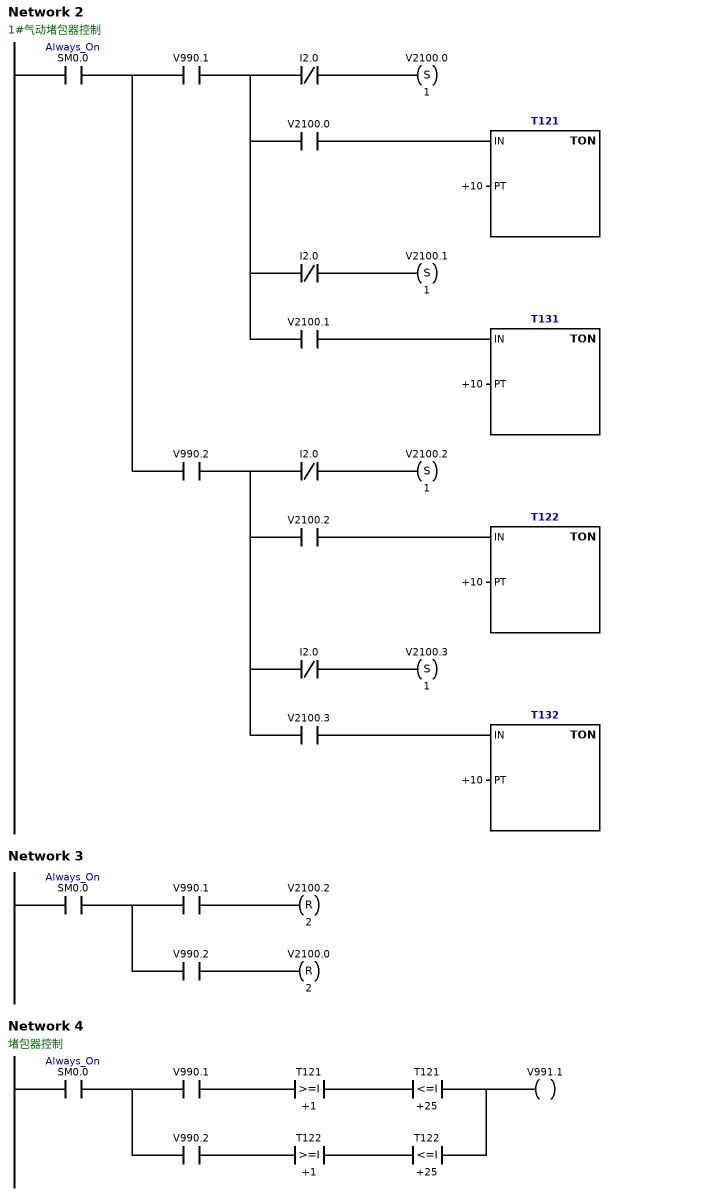
[picture p72: SBR29 networks 2-4]
Network 2
// 1#气动堵包器控制
LD     Always_On:SM0.0
LPS
A      V990.1
LPS
AN     I2.0
S      V2100.0, 1
LRD
A      V2100.0
TON    T121, +10
LRD
AN     I2.0
S      V2100.1, 1
LPP
A      V2100.1
TON    T131, +10
LPP
A      V990.2
LPS
AN     I2.0
S      V2100.2, 1
LRD
A      V2100.2
TON    T122, +10
LRD
AN     I2.0
S      V2100.3, 1
LPP
A      V2100.3
TON    T132, +10
Network 3
LD     Always_On:SM0.0
LPS
A      V990.1
R      V2100.2, 2
LPP
A      V990.2
R      V2100.0, 2
Network 4
// 堵包器控制
LD     Always_On:SM0.0
LD     V990.1
AW>=   T121, +1
AW<=   T121, +25
LD     V990.2
AW>=   T122, +1
AW<=   T122, +25
OLD
ALD
=      V991.1
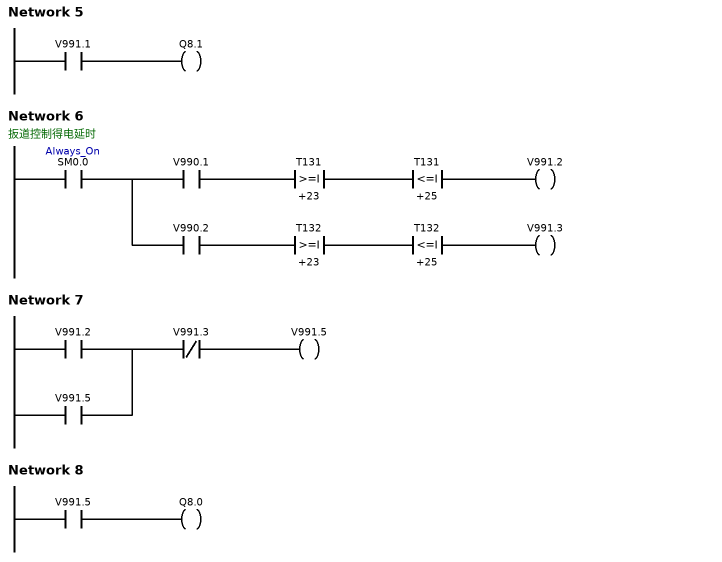
Network 5
LD     V991.1
=      Q8.1
Network 6
// 扳道控制得电延时
LD     Always_On:SM0.0
LPS
A      V990.1
AW>=   T131, +23
AW<=   T131, +25
=      V991.2
LPP
A      V990.2
AW>=   T132, +23
AW<=   T132, +25
=      V991.3
Network 7
LD     V991.2
O      V991.5
AN     V991.3
=      V991.5
Network 8
LD     V991.5
=      Q8.0
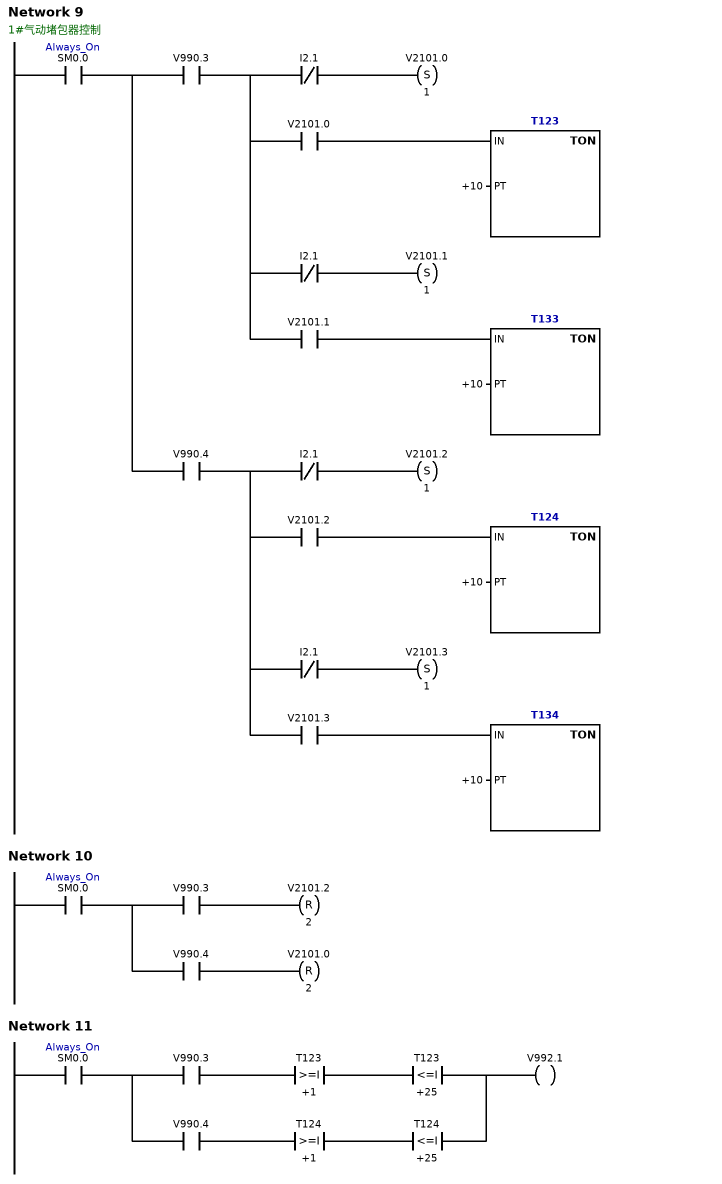
Network 9
// 1#气动堵包器控制
LD     Always_On:SM0.0
LPS
A      V990.3
LPS
AN     I2.1
S      V2101.0, 1
LRD
A      V2101.0
TON    T123, +10
LRD
AN     I2.1
S      V2101.1, 1
LPP
A      V2101.1
TON    T133, +10
LPP
A      V990.4
LPS
AN     I2.1
S      V2101.2, 1
LRD
A      V2101.2
TON    T124, +10
LRD
AN     I2.1
S      V2101.3, 1
LPP
A      V2101.3
TON    T134, +10
Network 10
LD     Always_On:SM0.0
LPS
A      V990.3
R      V2101.2, 2
LPP
A      V990.4
R      V2101.0, 2
Network 11
LD     Always_On:SM0.0
LD     V990.3
AW>=   T123, +1
AW<=   T123, +25
LD     V990.4
AW>=   T124, +1
AW<=   T124, +25
OLD
ALD
=      V992.1
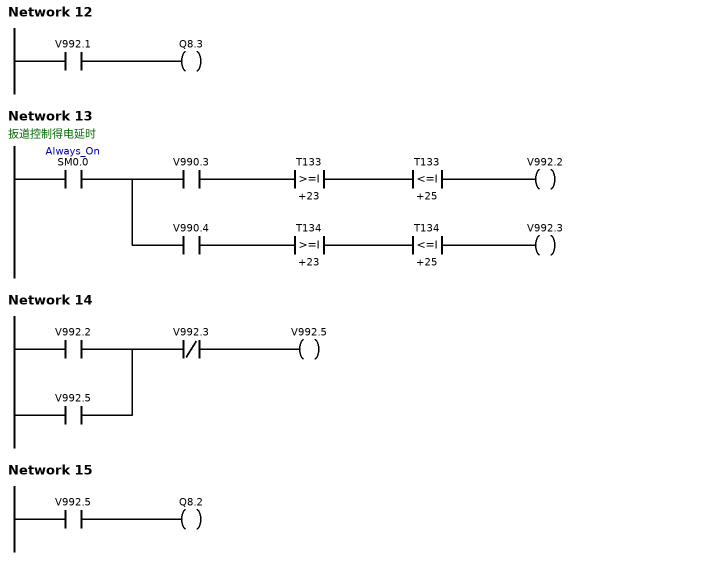
Network 12
LD     V992.1
=      Q8.3
Network 13
// 扳道控制得电延时
LD     Always_On:SM0.0
LPS
A      V990.3
AW>=   T133, +23
AW<=   T133, +25
=      V992.2
LPP
A      V990.4
AW>=   T134, +23
AW<=   T134, +25
=      V992.3
Network 14
LD     V992.2
O      V992.5
AN     V992.3
=      V992.5
Network 15
LD     V992.5
=      Q8.2
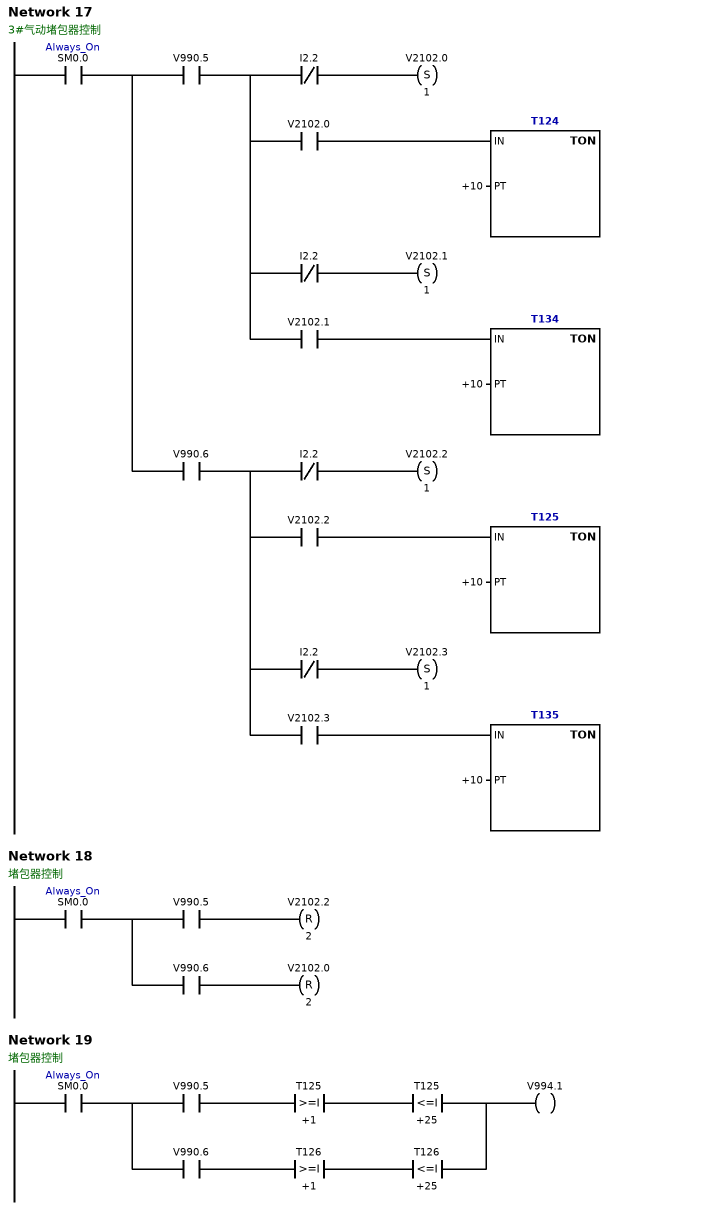
Network 17
// 3#气动堵包器控制
LD     Always_On:SM0.0
LPS
A      V990.5
LPS
AN     I2.2
S      V2102.0, 1
LRD
A      V2102.0
TON    T124, +10
LRD
AN     I2.2
S      V2102.1, 1
LPP
A      V2102.1
TON    T134, +10
LPP
A      V990.6
LPS
AN     I2.2
S      V2102.2, 1
LRD
A      V2102.2
TON    T125, +10
LRD
AN     I2.2
S      V2102.3, 1
LPP
A      V2102.3
TON    T135, +10
Network 18
// 堵包器控制
LD     Always_On:SM0.0
LPS
A      V990.5
R      V2102.2, 2
LPP
A      V990.6
R      V2102.0, 2
Network 19
// 堵包器控制
LD     Always_On:SM0.0
LD     V990.5
AW>=   T125, +1
AW<=   T125, +25
LD     V990.6
AW>=   T126, +1
AW<=   T126, +25
OLD
ALD
=      V994.1
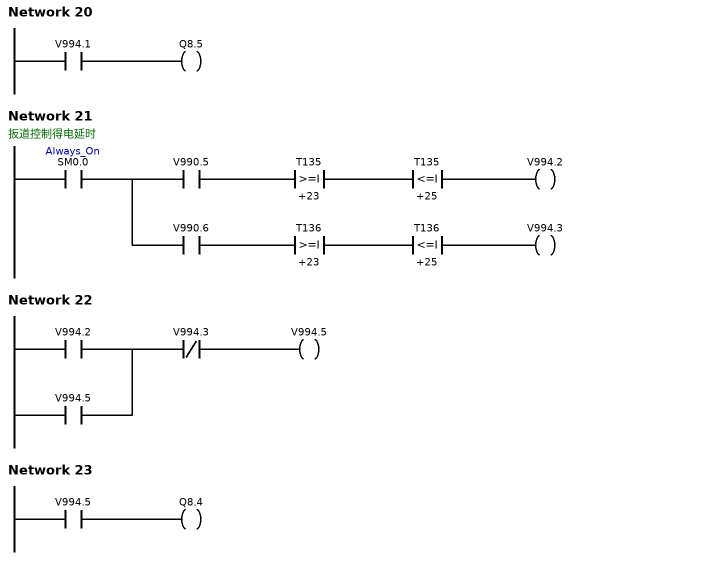
Network 20
LD     V994.1
=      Q8.5
Network 21
// 扳道控制得电延时
LD     Always_On:SM0.0
LPS
A      V990.5
AW>=   T135, +23
AW<=   T135, +25
=      V994.2
LPP
A      V990.6
AW>=   T136, +23
AW<=   T136, +25
=      V994.3
Network 22
LD     V994.2
O      V994.5
AN     V994.3
=      V994.5
Network 23
LD     V994.5
=      Q8.4
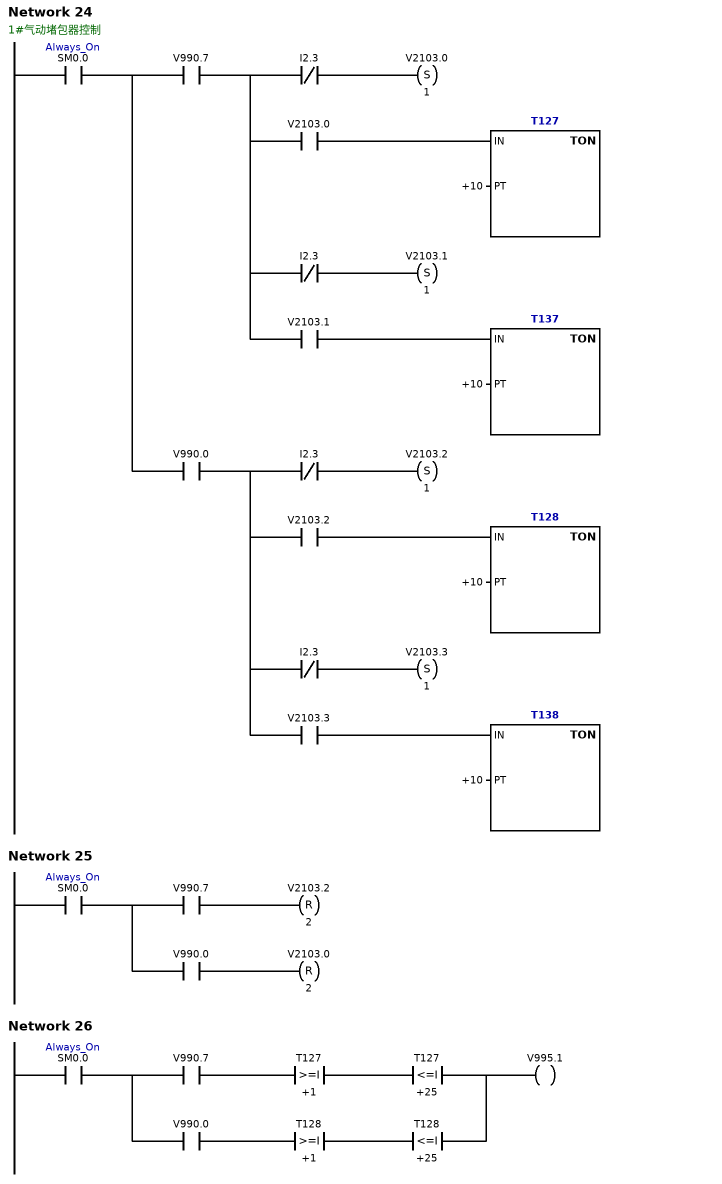
Network 24
// 1#气动堵包器控制
LD     Always_On:SM0.0
LPS
A      V990.7
LPS
AN     I2.3
S      V2103.0, 1
LRD
A      V2103.0
TON    T127, +10
LRD
AN     I2.3
S      V2103.1, 1
LPP
A      V2103.1
TON    T137, +10
LPP
A      V990.0
LPS
AN     I2.3
S      V2103.2, 1
LRD
A      V2103.2
TON    T128, +10
LRD
AN     I2.3
S      V2103.3, 1
LPP
A      V2103.3
TON    T138, +10
Network 25
LD     Always_On:SM0.0
LPS
A      V990.7
R      V2103.2, 2
LPP
A      V990.0
R      V2103.0, 2
Network 26
LD     Always_On:SM0.0
LD     V990.7
AW>=   T127, +1
AW<=   T127, +25
LD     V990.0
AW>=   T128, +1
AW<=   T128, +25
OLD
ALD
=      V995.1
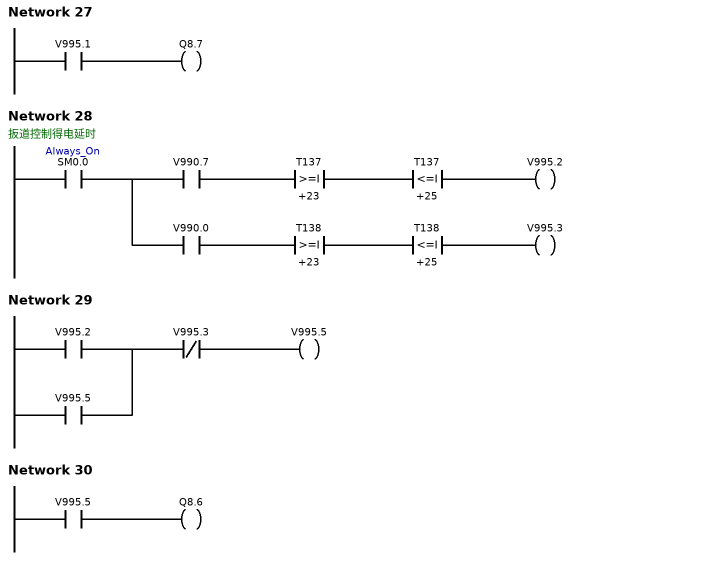
Network 27
LD     V995.1
=      Q8.7
Network 28
// 扳道控制得电延时
LD     Always_On:SM0.0
LPS
A      V990.7
AW>=   T137, +23
AW<=   T137, +25
=      V995.2
LPP
A      V990.0
AW>=   T138, +23
AW<=   T138, +25
=      V995.3
Network 29
LD     V995.2
O      V995.5
AN     V995.3
=      V995.5
Network 30
LD     V995.5
=      Q8.6
END_SUBROUTINE_BLOCK

SUBROUTINE_BLOCK GGLED1_2:SBR31
TITLE=子程序注释
VAR_INPUT
屏3地址:BYTE;	// LB0 
END_VAR
BEGIN
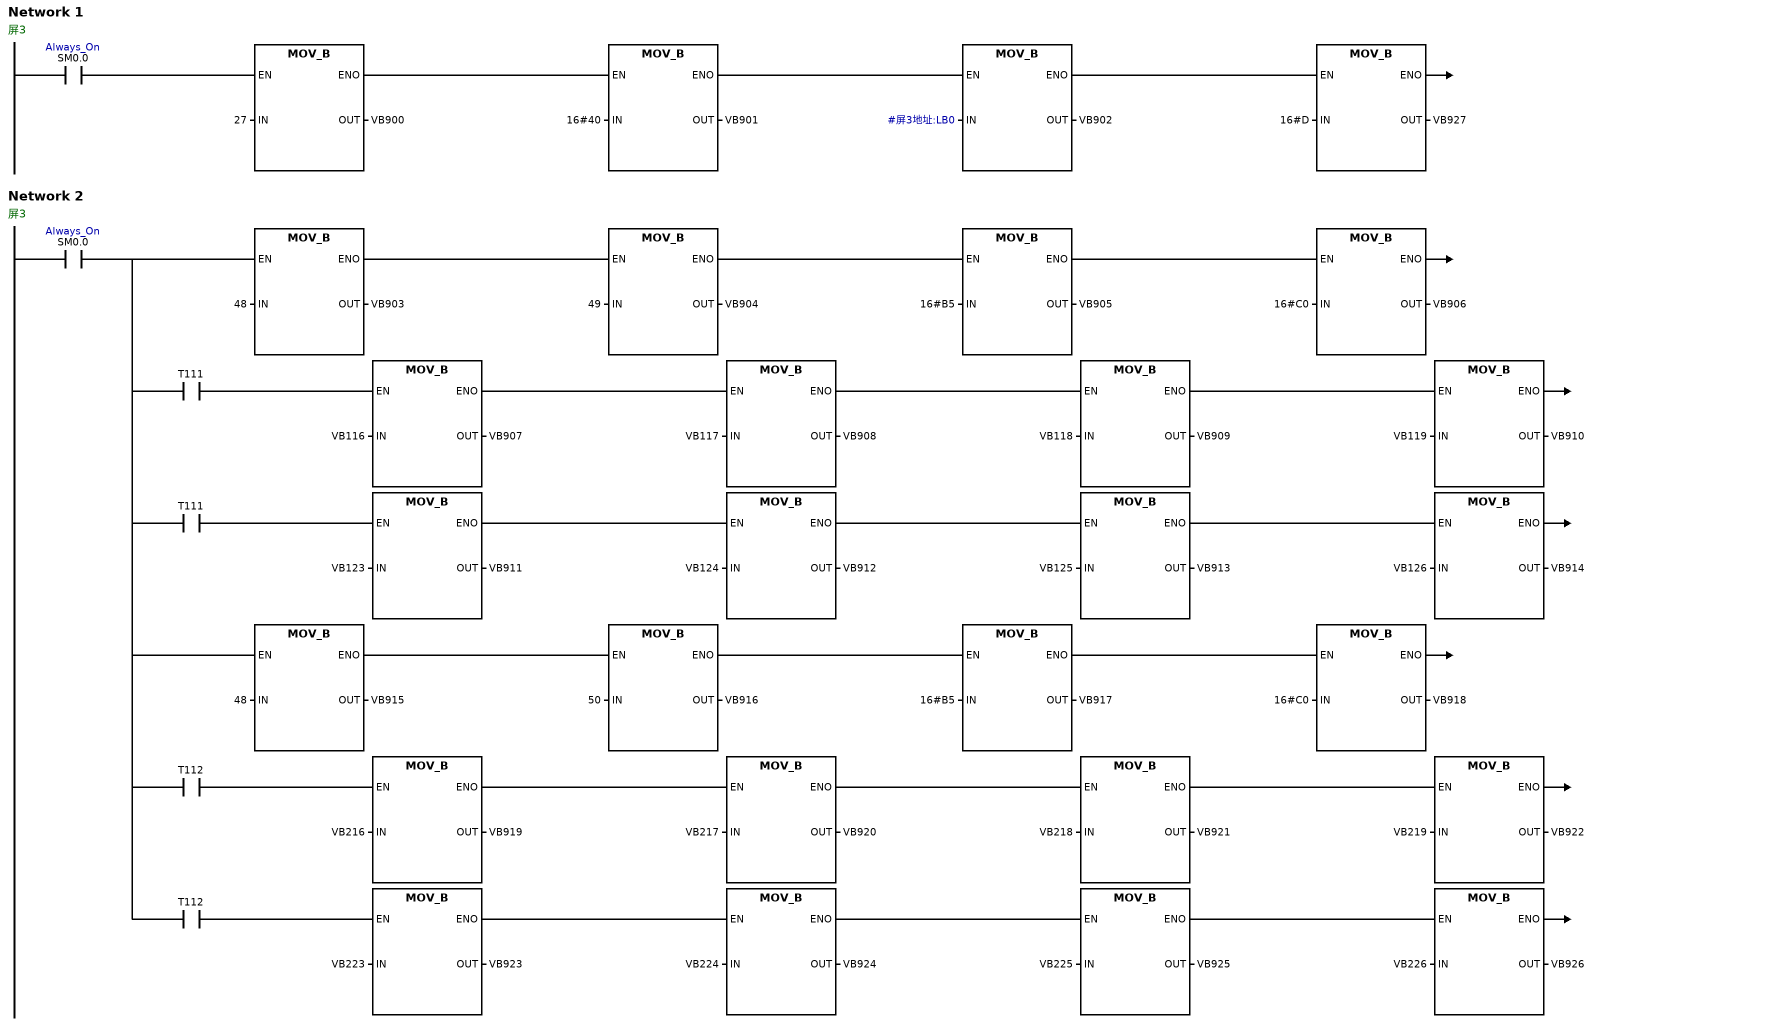
Network 1
// 屏3
LD     Always_On:SM0.0
MOVB   27, VB900
AENO
MOVB   16#40, VB901
AENO
MOVB   #屏3地址:LB0, VB902
AENO
MOVB   16#D, VB927
Network 2
// 屏3
LD     Always_On:SM0.0
LPS
MOVB   48, VB903
AENO
MOVB   49, VB904
AENO
MOVB   16#B5, VB905
AENO
MOVB   16#C0, VB906
LRD
A      T111
MOVB   VB116, VB907
AENO
MOVB   VB117, VB908
AENO
MOVB   VB118, VB909
AENO
MOVB   VB119, VB910
LRD
A      T111
MOVB   VB123, VB911
AENO
MOVB   VB124, VB912
AENO
MOVB   VB125, VB913
AENO
MOVB   VB126, VB914
LRD
MOVB   48, VB915
AENO
MOVB   50, VB916
AENO
MOVB   16#B5, VB917
AENO
MOVB   16#C0, VB918
LRD
A      T112
MOVB   VB216, VB919
AENO
MOVB   VB217, VB920
AENO
MOVB   VB218, VB921
AENO
MOVB   VB219, VB922
LPP
A      T112
MOVB   VB223, VB923
AENO
MOVB   VB224, VB924
AENO
MOVB   VB225, VB925
AENO
MOVB   VB226, VB926
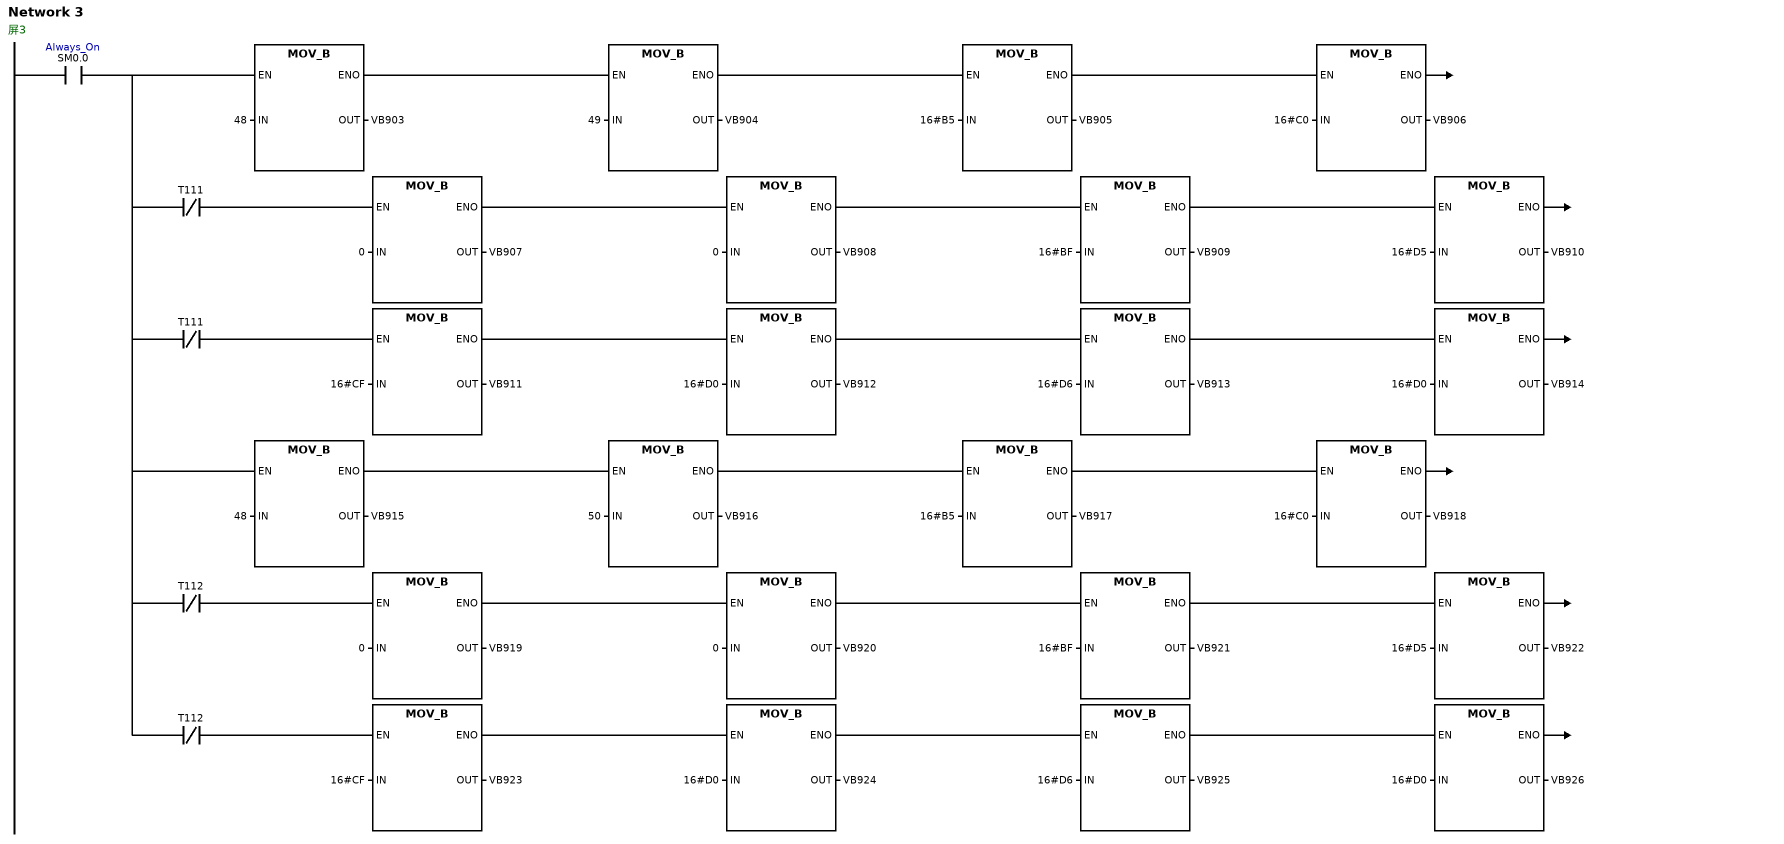
Network 3
// 屏3
LD     Always_On:SM0.0
LPS
MOVB   48, VB903
AENO
MOVB   49, VB904
AENO
MOVB   16#B5, VB905
AENO
MOVB   16#C0, VB906
LRD
AN     T111
MOVB   0, VB907
AENO
MOVB   0, VB908
AENO
MOVB   16#BF, VB909
AENO
MOVB   16#D5, VB910
LRD
AN     T111
MOVB   16#CF, VB911
AENO
MOVB   16#D0, VB912
AENO
MOVB   16#D6, VB913
AENO
MOVB   16#D0, VB914
LRD
MOVB   48, VB915
AENO
MOVB   50, VB916
AENO
MOVB   16#B5, VB917
AENO
MOVB   16#C0, VB918
LRD
AN     T112
MOVB   0, VB919
AENO
MOVB   0, VB920
AENO
MOVB   16#BF, VB921
AENO
MOVB   16#D5, VB922
LPP
AN     T112
MOVB   16#CF, VB923
AENO
MOVB   16#D0, VB924
AENO
MOVB   16#D6, VB925
AENO
MOVB   16#D0, VB926
END_SUBROUTINE_BLOCK

SUBROUTINE_BLOCK GGLED3_4:SBR32
TITLE=子程序注释
VAR_INPUT
屏3地址:BYTE;	// LB0 
END_VAR
BEGIN
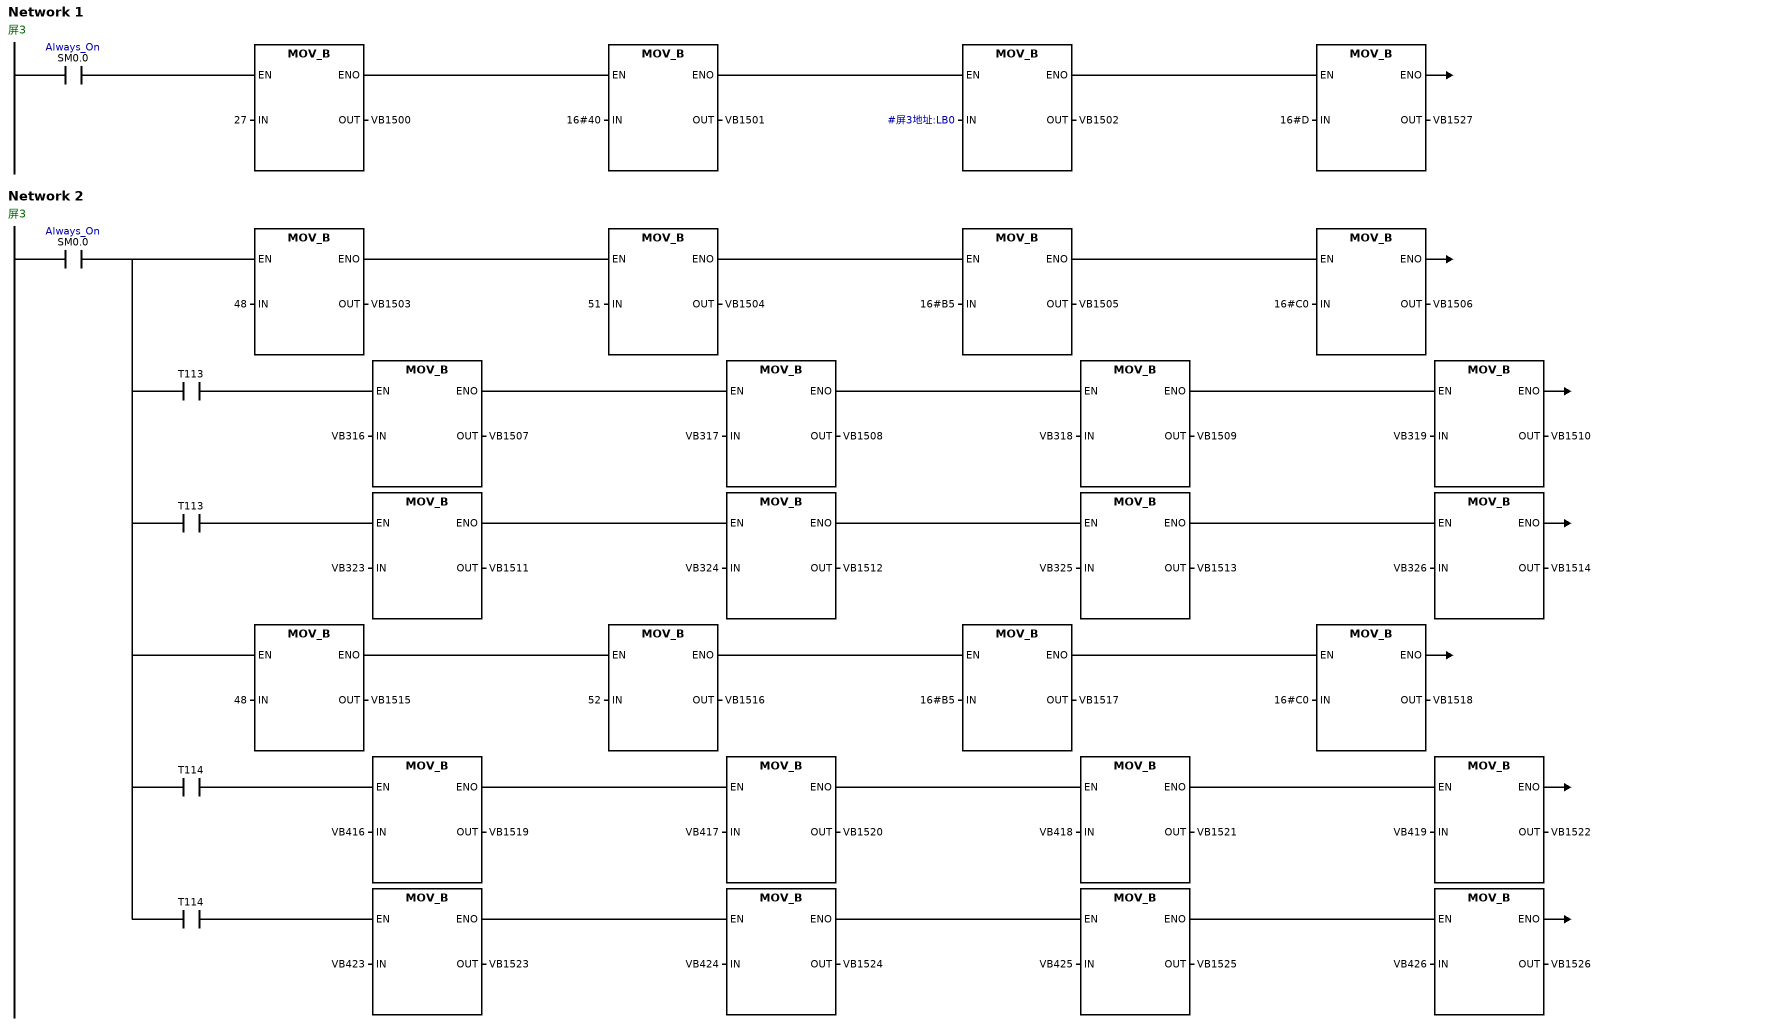
Network 1
// 屏3
LD     Always_On:SM0.0
MOVB   27, VB1500
AENO
MOVB   16#40, VB1501
AENO
MOVB   #屏3地址:LB0, VB1502
AENO
MOVB   16#D, VB1527
Network 2
// 屏3
LD     Always_On:SM0.0
LPS
MOVB   48, VB1503
AENO
MOVB   51, VB1504
AENO
MOVB   16#B5, VB1505
AENO
MOVB   16#C0, VB1506
LRD
A      T113
MOVB   VB316, VB1507
AENO
MOVB   VB317, VB1508
AENO
MOVB   VB318, VB1509
AENO
MOVB   VB319, VB1510
LRD
A      T113
MOVB   VB323, VB1511
AENO
MOVB   VB324, VB1512
AENO
MOVB   VB325, VB1513
AENO
MOVB   VB326, VB1514
LRD
MOVB   48, VB1515
AENO
MOVB   52, VB1516
AENO
MOVB   16#B5, VB1517
AENO
MOVB   16#C0, VB1518
LRD
A      T114
MOVB   VB416, VB1519
AENO
MOVB   VB417, VB1520
AENO
MOVB   VB418, VB1521
AENO
MOVB   VB419, VB1522
LPP
A      T114
MOVB   VB423, VB1523
AENO
MOVB   VB424, VB1524
AENO
MOVB   VB425, VB1525
AENO
MOVB   VB426, VB1526
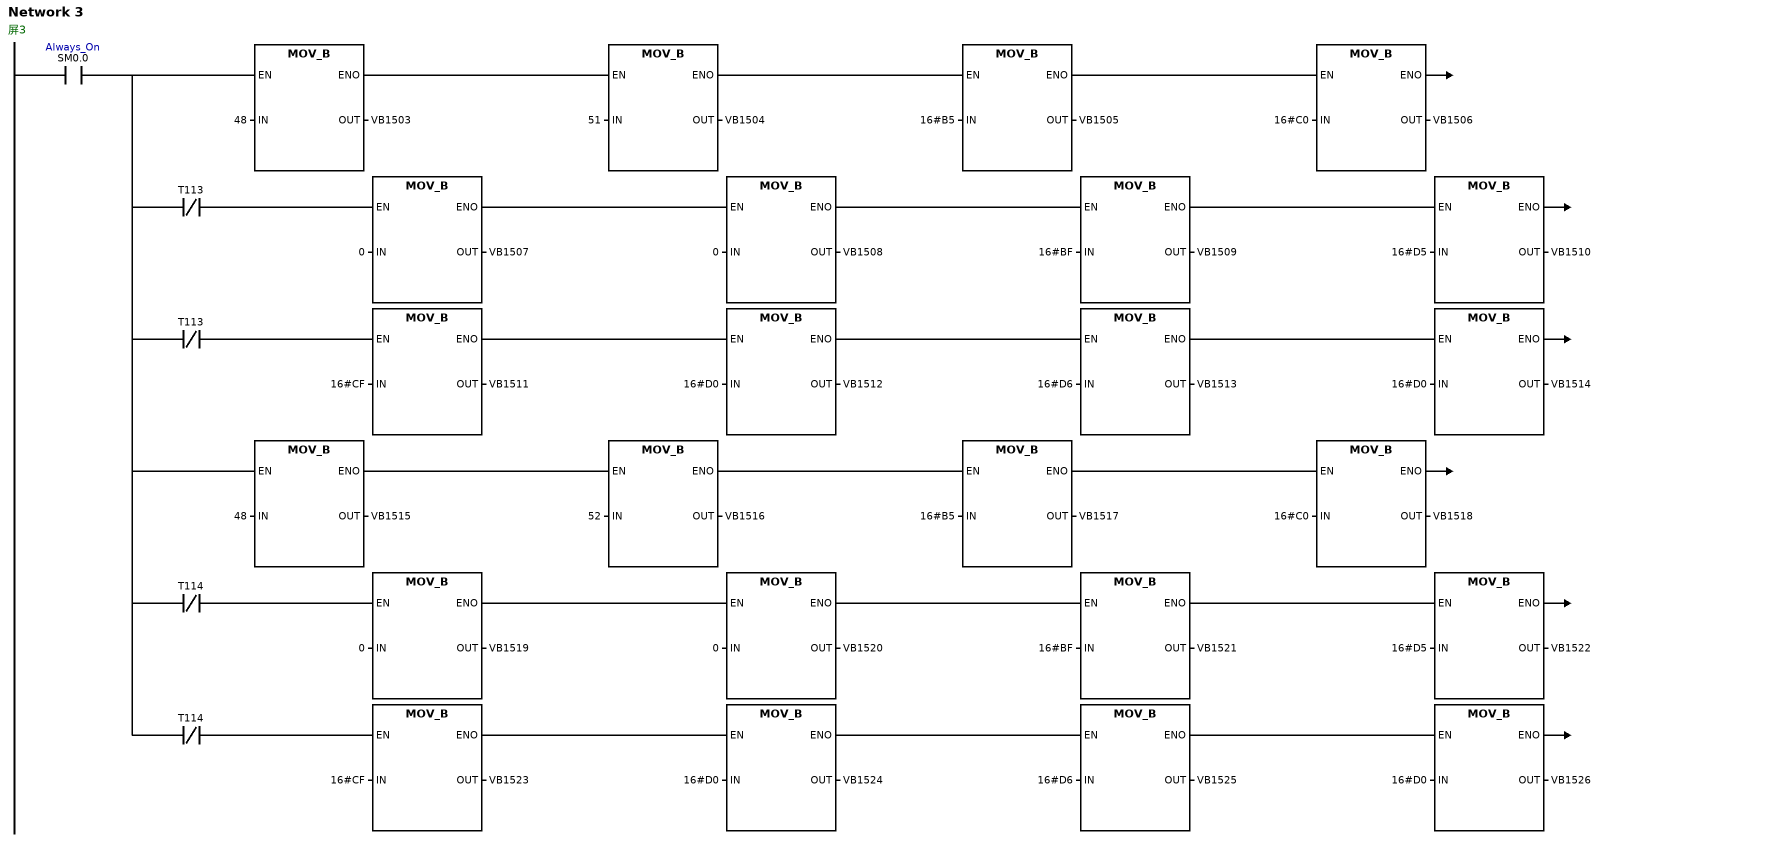
Network 3
// 屏3
LD     Always_On:SM0.0
LPS
MOVB   48, VB1503
AENO
MOVB   51, VB1504
AENO
MOVB   16#B5, VB1505
AENO
MOVB   16#C0, VB1506
LRD
AN     T113
MOVB   0, VB1507
AENO
MOVB   0, VB1508
AENO
MOVB   16#BF, VB1509
AENO
MOVB   16#D5, VB1510
LRD
AN     T113
MOVB   16#CF, VB1511
AENO
MOVB   16#D0, VB1512
AENO
MOVB   16#D6, VB1513
AENO
MOVB   16#D0, VB1514
LRD
MOVB   48, VB1515
AENO
MOVB   52, VB1516
AENO
MOVB   16#B5, VB1517
AENO
MOVB   16#C0, VB1518
LRD
AN     T114
MOVB   0, VB1519
AENO
MOVB   0, VB1520
AENO
MOVB   16#BF, VB1521
AENO
MOVB   16#D5, VB1522
LPP
AN     T114
MOVB   16#CF, VB1523
AENO
MOVB   16#D0, VB1524
AENO
MOVB   16#D6, VB1525
AENO
MOVB   16#D0, VB1526
END_SUBROUTINE_BLOCK

SUBROUTINE_BLOCK GGLED5_6:SBR33
TITLE=子程序注释
VAR_INPUT
屏3地址:BYTE;	// LB0 
END_VAR
BEGIN
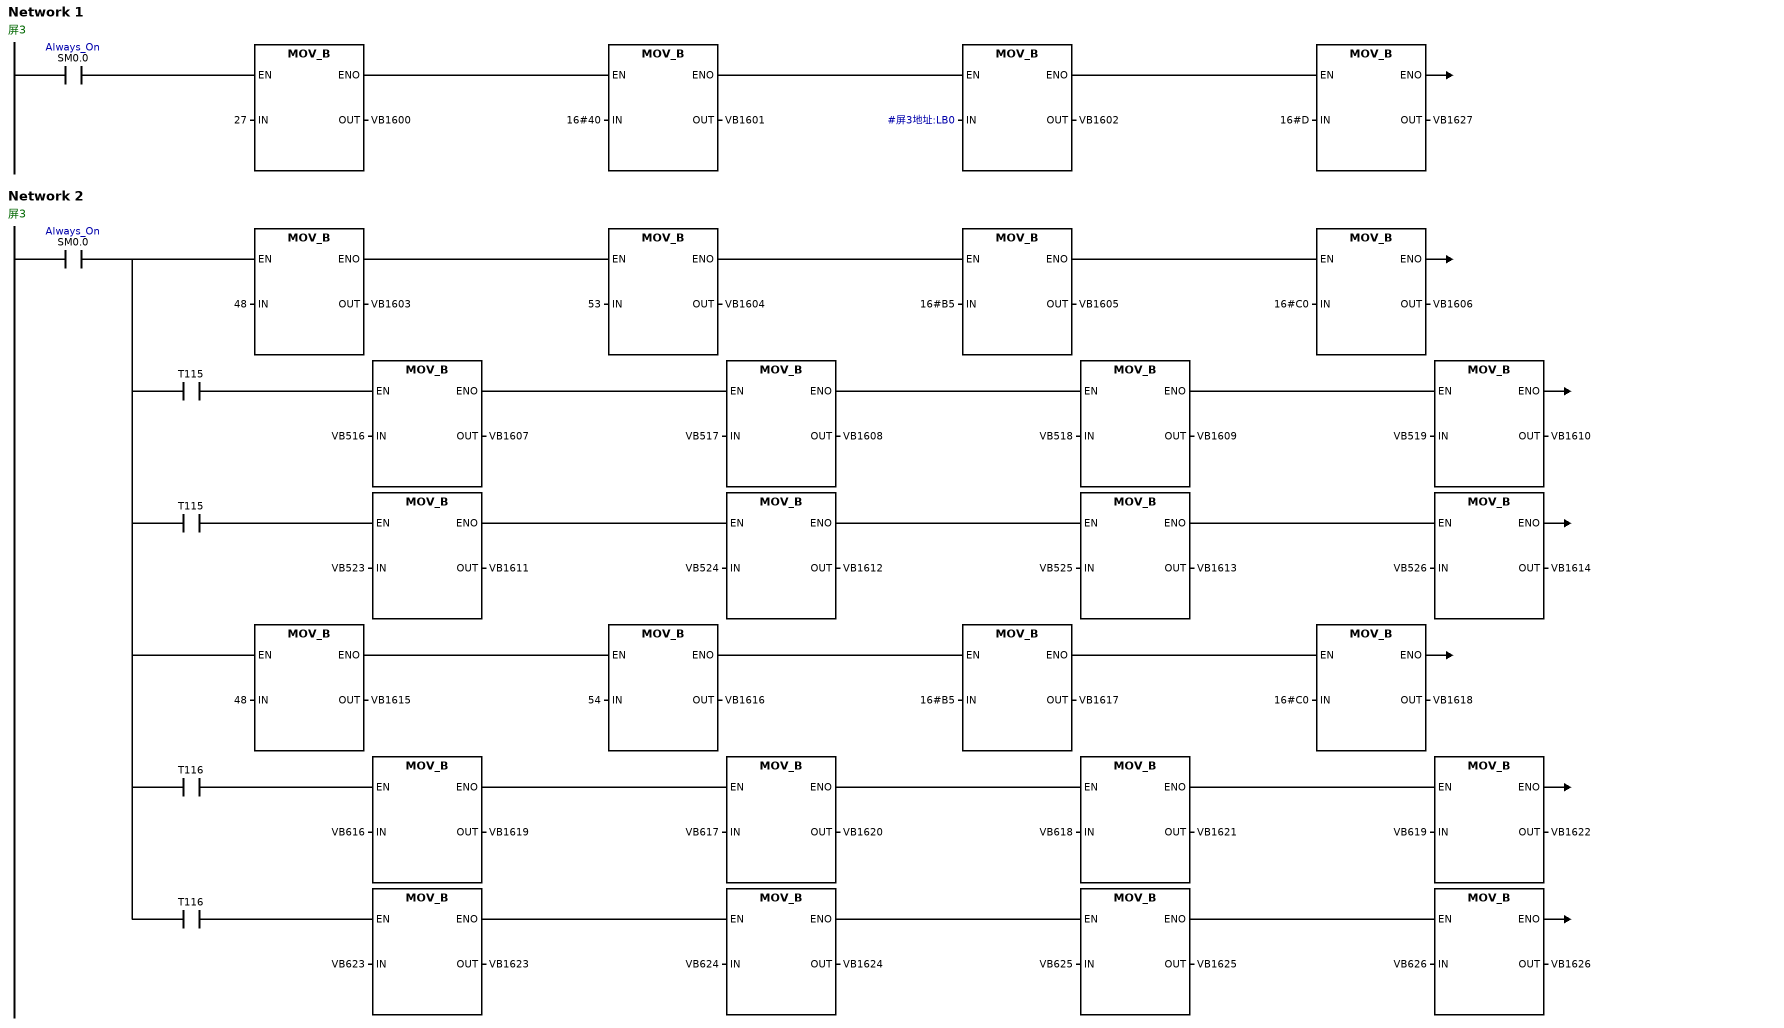
Network 1
// 屏3
LD     Always_On:SM0.0
MOVB   27, VB1600
AENO
MOVB   16#40, VB1601
AENO
MOVB   #屏3地址:LB0, VB1602
AENO
MOVB   16#D, VB1627
Network 2
// 屏3
LD     Always_On:SM0.0
LPS
MOVB   48, VB1603
AENO
MOVB   53, VB1604
AENO
MOVB   16#B5, VB1605
AENO
MOVB   16#C0, VB1606
LRD
A      T115
MOVB   VB516, VB1607
AENO
MOVB   VB517, VB1608
AENO
MOVB   VB518, VB1609
AENO
MOVB   VB519, VB1610
LRD
A      T115
MOVB   VB523, VB1611
AENO
MOVB   VB524, VB1612
AENO
MOVB   VB525, VB1613
AENO
MOVB   VB526, VB1614
LRD
MOVB   48, VB1615
AENO
MOVB   54, VB1616
AENO
MOVB   16#B5, VB1617
AENO
MOVB   16#C0, VB1618
LRD
A      T116
MOVB   VB616, VB1619
AENO
MOVB   VB617, VB1620
AENO
MOVB   VB618, VB1621
AENO
MOVB   VB619, VB1622
LPP
A      T116
MOVB   VB623, VB1623
AENO
MOVB   VB624, VB1624
AENO
MOVB   VB625, VB1625
AENO
MOVB   VB626, VB1626
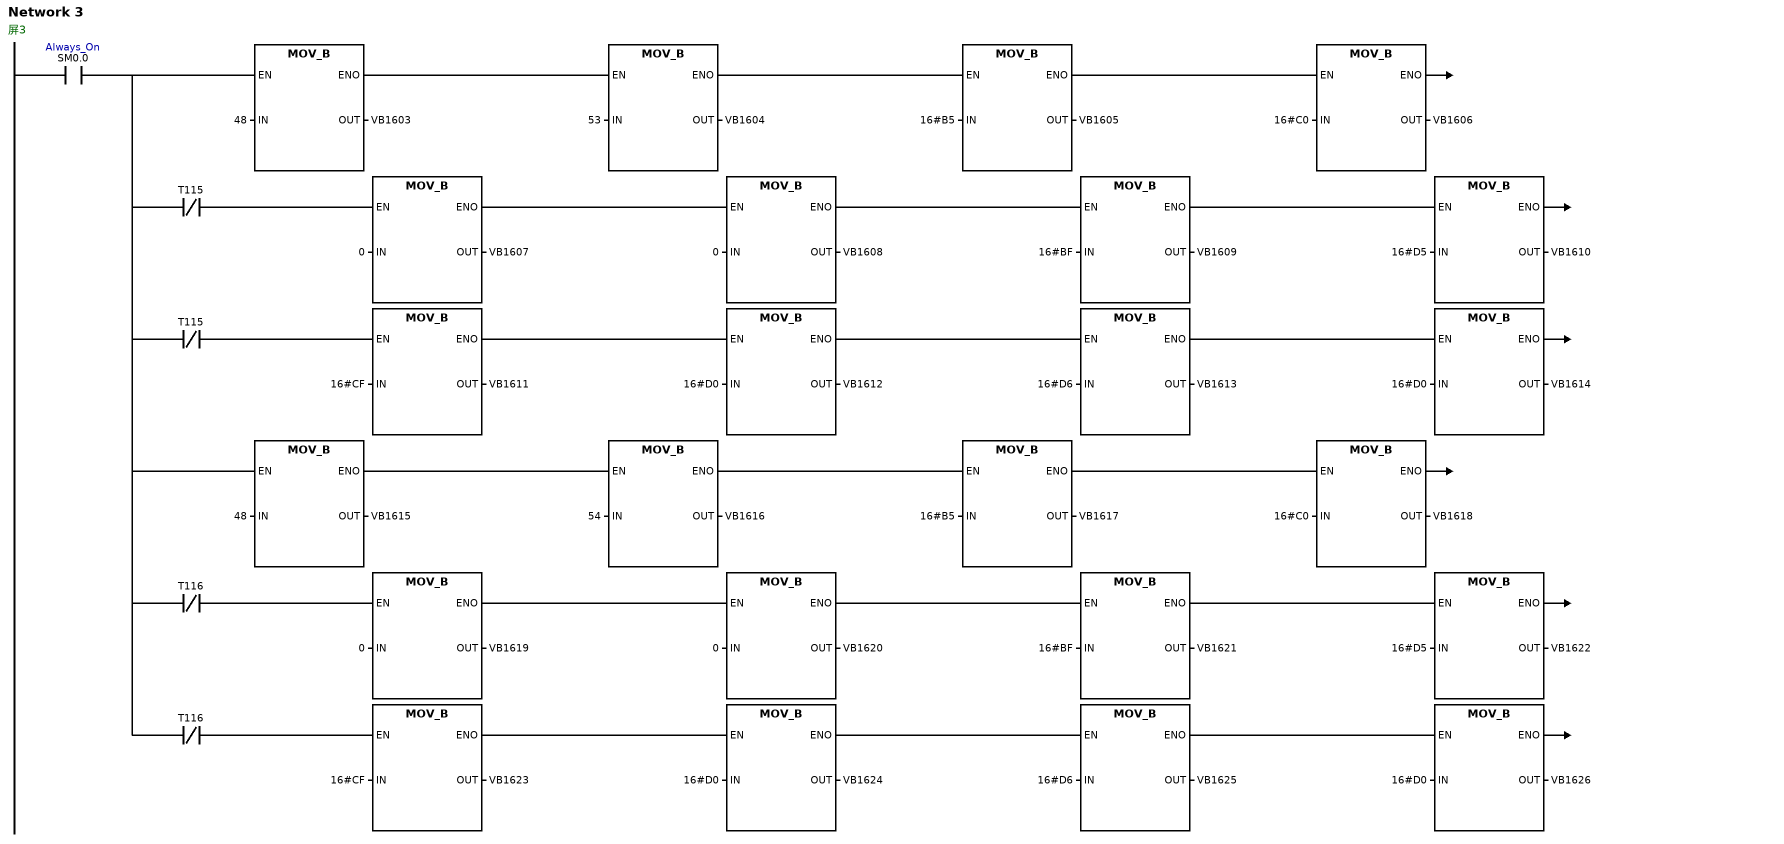
Network 3
// 屏3
LD     Always_On:SM0.0
LPS
MOVB   48, VB1603
AENO
MOVB   53, VB1604
AENO
MOVB   16#B5, VB1605
AENO
MOVB   16#C0, VB1606
LRD
AN     T115
MOVB   0, VB1607
AENO
MOVB   0, VB1608
AENO
MOVB   16#BF, VB1609
AENO
MOVB   16#D5, VB1610
LRD
AN     T115
MOVB   16#CF, VB1611
AENO
MOVB   16#D0, VB1612
AENO
MOVB   16#D6, VB1613
AENO
MOVB   16#D0, VB1614
LRD
MOVB   48, VB1615
AENO
MOVB   54, VB1616
AENO
MOVB   16#B5, VB1617
AENO
MOVB   16#C0, VB1618
LRD
AN     T116
MOVB   0, VB1619
AENO
MOVB   0, VB1620
AENO
MOVB   16#BF, VB1621
AENO
MOVB   16#D5, VB1622
LPP
AN     T116
MOVB   16#CF, VB1623
AENO
MOVB   16#D0, VB1624
AENO
MOVB   16#D6, VB1625
AENO
MOVB   16#D0, VB1626
END_SUBROUTINE_BLOCK

SUBROUTINE_BLOCK GGLED7_8:SBR34
TITLE=子程序注释
VAR_INPUT
屏3地址:BYTE;	// LB0 
END_VAR
BEGIN
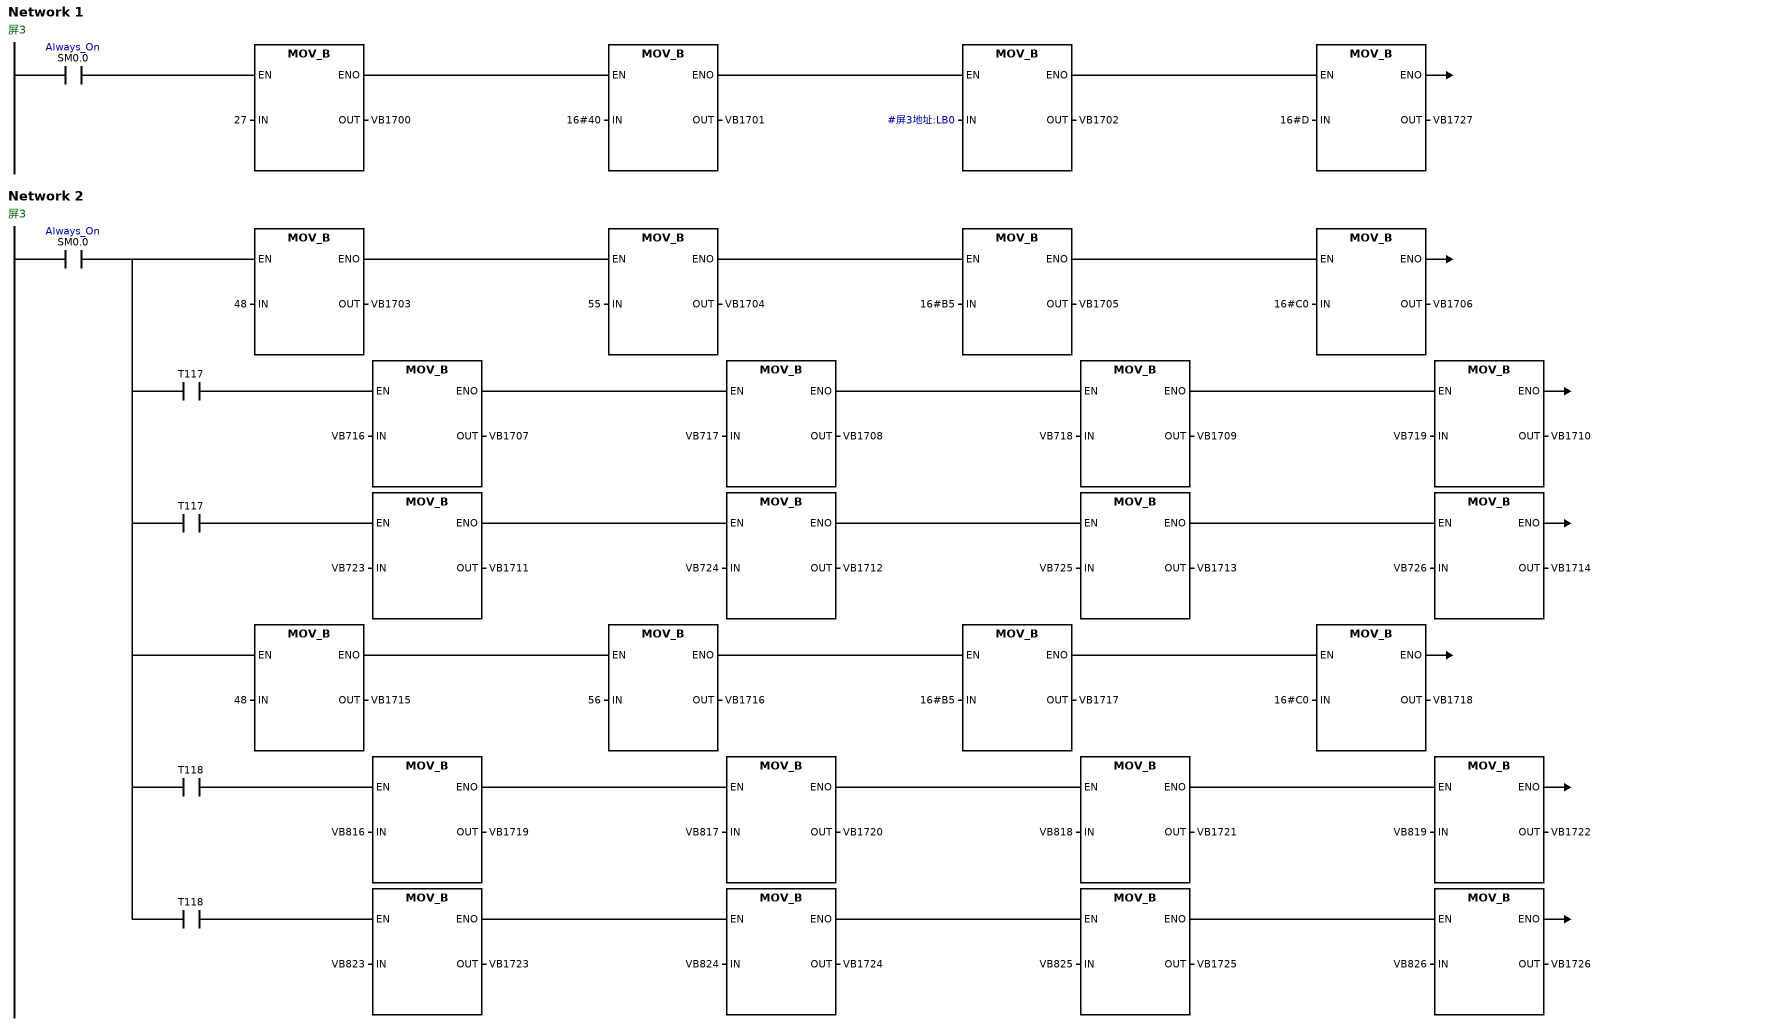
Network 1
// 屏3
LD     Always_On:SM0.0
MOVB   27, VB1700
AENO
MOVB   16#40, VB1701
AENO
MOVB   #屏3地址:LB0, VB1702
AENO
MOVB   16#D, VB1727
Network 2
// 屏3
LD     Always_On:SM0.0
LPS
MOVB   48, VB1703
AENO
MOVB   55, VB1704
AENO
MOVB   16#B5, VB1705
AENO
MOVB   16#C0, VB1706
LRD
A      T117
MOVB   VB716, VB1707
AENO
MOVB   VB717, VB1708
AENO
MOVB   VB718, VB1709
AENO
MOVB   VB719, VB1710
LRD
A      T117
MOVB   VB723, VB1711
AENO
MOVB   VB724, VB1712
AENO
MOVB   VB725, VB1713
AENO
MOVB   VB726, VB1714
LRD
MOVB   48, VB1715
AENO
MOVB   56, VB1716
AENO
MOVB   16#B5, VB1717
AENO
MOVB   16#C0, VB1718
LRD
A      T118
MOVB   VB816, VB1719
AENO
MOVB   VB817, VB1720
AENO
MOVB   VB818, VB1721
AENO
MOVB   VB819, VB1722
LPP
A      T118
MOVB   VB823, VB1723
AENO
MOVB   VB824, VB1724
AENO
MOVB   VB825, VB1725
AENO
MOVB   VB826, VB1726
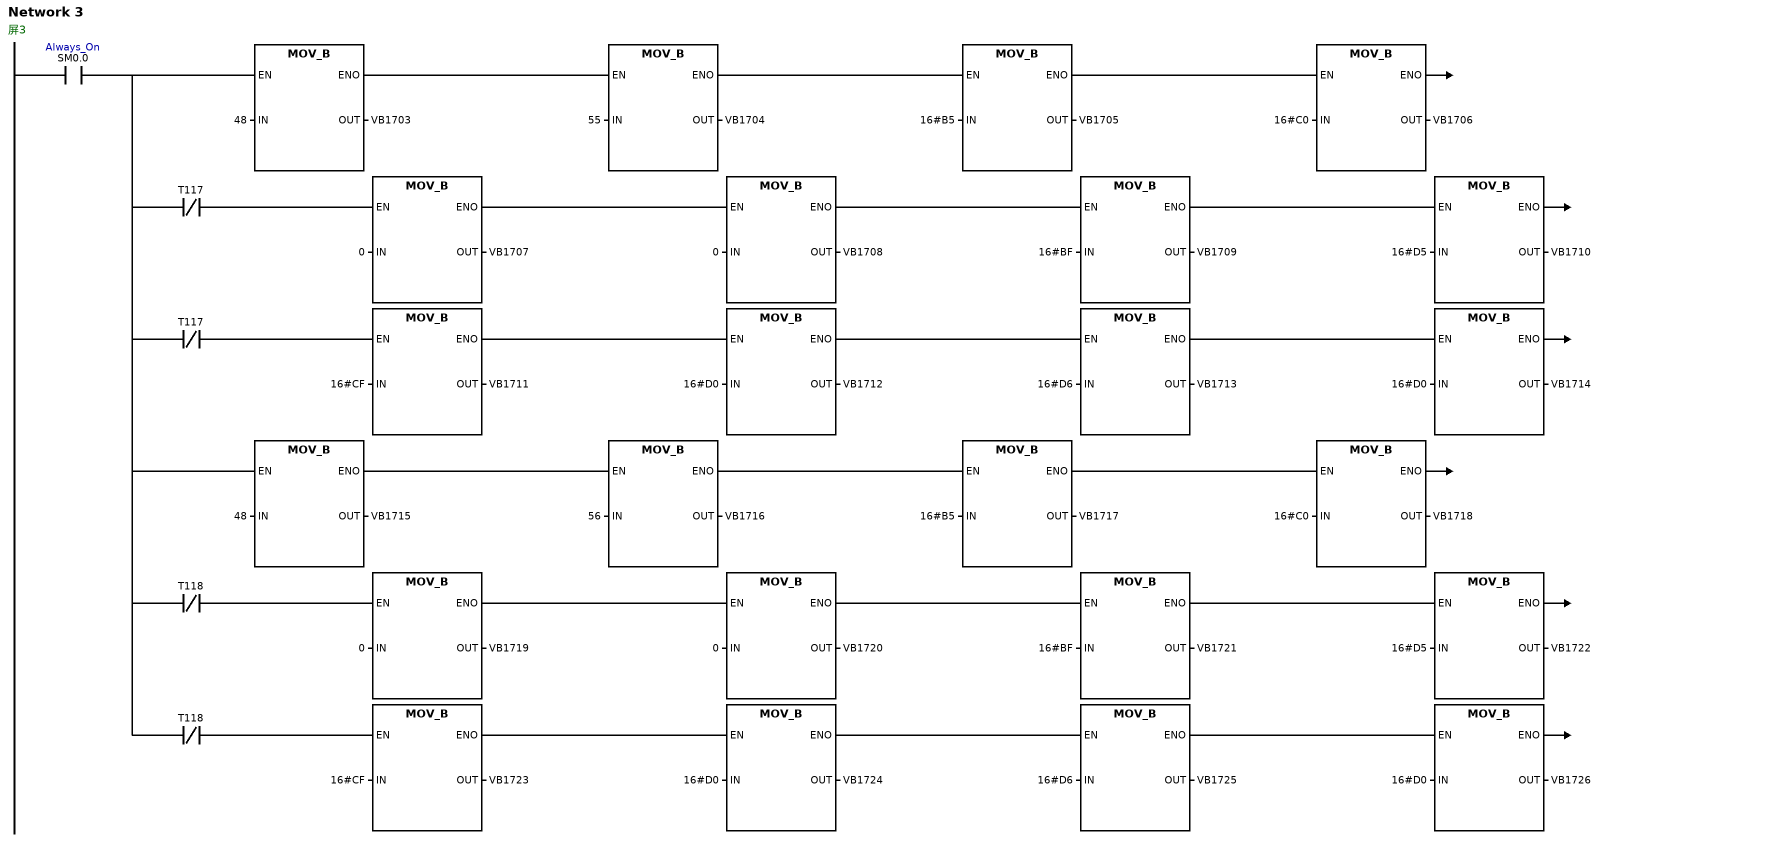
Network 3
// 屏3
LD     Always_On:SM0.0
LPS
MOVB   48, VB1703
AENO
MOVB   55, VB1704
AENO
MOVB   16#B5, VB1705
AENO
MOVB   16#C0, VB1706
LRD
AN     T117
MOVB   0, VB1707
AENO
MOVB   0, VB1708
AENO
MOVB   16#BF, VB1709
AENO
MOVB   16#D5, VB1710
LRD
AN     T117
MOVB   16#CF, VB1711
AENO
MOVB   16#D0, VB1712
AENO
MOVB   16#D6, VB1713
AENO
MOVB   16#D0, VB1714
LRD
MOVB   48, VB1715
AENO
MOVB   56, VB1716
AENO
MOVB   16#B5, VB1717
AENO
MOVB   16#C0, VB1718
LRD
AN     T118
MOVB   0, VB1719
AENO
MOVB   0, VB1720
AENO
MOVB   16#BF, VB1721
AENO
MOVB   16#D5, VB1722
LPP
AN     T118
MOVB   16#CF, VB1723
AENO
MOVB   16#D0, VB1724
AENO
MOVB   16#D6, VB1725
AENO
MOVB   16#D0, VB1726
END_SUBROUTINE_BLOCK

// SBR80: protected block, not included

// SBR81: protected block, not included

// SBR82: protected block, not included

// SBR85: protected block, not included
